FUNCTION_BLOCK 1D_MOVETO_PARALLEL_PLANE
  (* Standard: 61499-2 *)
  (* Version 1.0, 22-03-12, GASR, Universidade do Estado de Santa Catarina *)
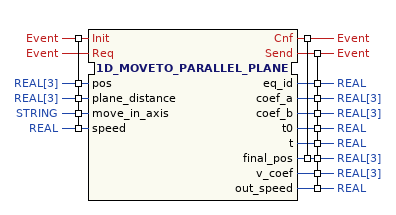
  EVENT_INPUT
    Init WITH pos, plane_distance, move_in_axis, speed; (* Initialization request *)
    Req; (* Requisition to finish *)
  END_EVENT
  EVENT_OUTPUT
    Cnf WITH final_pos; (* Execution Confirmed *)
    Send WITH eq_id, coef_a, coef_b, t0, t, final_pos, out_speed, v_coef; (* Send data *)
  END_EVENT
  VAR_INPUT
    pos : ARRAY [0..2] OF REAL; (* Machine position *)
    plane_distance : ARRAY [0..2] OF REAL; (* Security plane position *)
    move_in_axis : STRING; (* 'x', 'y' or 'z' *)
    speed : REAL := 0; (* Feedrate in m/s *)
  END_VAR
  VAR_OUTPUT
    eq_id : REAL; (* Curve equation id *)
    coef_a : ARRAY [0..2] OF REAL; (* Line angular coeficient *)
    coef_b : ARRAY [0..2] OF REAL; (* Line linear coeficient *)
    t0 : REAL; (* Initial parameter *)
    t : REAL; (* Final parameter *)
    final_pos : ARRAY [0..2] OF REAL; (* Final position *)
    v_coef : ARRAY [0..2] OF REAL; (* Velocity coeficient *)
    out_speed : REAL; (* Speed in m/s *)
  END_VAR
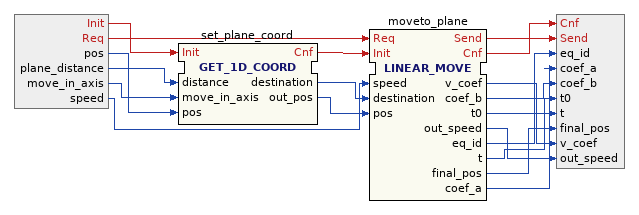
  FBS
    set_plane_coord : GET_1D_COORD;
    moveto_plane : LINEAR_MOVE;
  END_FBS
  EVENT_CONNECTIONS
    Req TO moveto_plane.Req;
    Init TO set_plane_coord.Init;
    set_plane_coord.Cnf TO moveto_plane.Init;
    moveto_plane.Send TO Send;
    moveto_plane.Cnf TO Cnf;
  END_CONNECTIONS
  DATA_CONNECTIONS
    moveto_plane.v_coef TO v_coef;
    moveto_plane.coef_b TO coef_b;
    moveto_plane.t0 TO t0;
    moveto_plane.out_speed TO out_speed;
    moveto_plane.eq_id TO eq_id;
    moveto_plane.t TO t;
    moveto_plane.final_pos TO final_pos;
    moveto_plane.coef_a TO coef_a;
    plane_distance TO set_plane_coord.distance;
    move_in_axis TO set_plane_coord.move_in_axis;
    pos TO set_plane_coord.pos;
    speed TO moveto_plane.speed;
    set_plane_coord.destination TO moveto_plane.destination;
    set_plane_coord.out_pos TO moveto_plane.pos;
  END_CONNECTIONS
END_FUNCTION_BLOCK
